TYPE ST_ProcessStationStatus :
STRUCT
    eState                    : E_ProcessStationState;
    eFault                    : E_ProcessStationFault;
    bReady                    : BOOL;
    bBusy                     : BOOL;
    bFaulted                  : BOOL;
    bSafePosition             : BOOL;
    bCylinderExtended         : BOOL;
    bCylinderRetracted        : BOOL;
    bExtendPermissive         : BOOL;
    bRetractPermissive        : BOOL;
    bAutomaticRequestActive   : BOOL;
    bManualRequestActive      : BOOL;
    bEquipmentReady           : BOOL;
    bEquipmentBusy            : BOOL;
    bEquipmentFaulted         : BOOL;
    sMessage                  : STRING(160);
END_STRUCT
END_TYPE

(* stored: Version 1.1.0.1, ProductVersion 3.1.4026.18
   DUT ST_ProcessStationStatus: Id {8680f870-eff6-4a86-9523-398081b6870f} *)
